{attribute addProperty BoxType "EL6201-0000-0017"}
{attribute addProperty Id "Slave_1_OutputsAT %Q*Slave_1_Outputs_44535924811Slave_2_OutputsAT %Q*Slave_2_Outputs_DA85B14E819Slave_3_OutputsAT %Q*Slave_3_Outputs_6031563F8117Slave_4_OutputsAT %Q*Slave_4_Outputs_A2C52F8B8125Slave_5_OutputsAT %Q*Slave_5_Outputs_502A55918133Slave_6_OutputsAT %Q*Slave_6_Outputs_564C8B0F8141Slave_7_OutputsAT %Q*Slave_7_Outputs_0A95F91A8149Slave_8_OutputsAT %Q*Slave_8_Outputs_C94C3BE28157Slave_9_OutputsAT %Q*Slave_9_Outputs_10CA7D998165Slave_10_OutputsAT %Q*Slave_10_Outputs_BCBE3A9D8173Slave_11_OutputsAT %Q*Slave_11_Outputs_22455BE68181Slave_12_OutputsAT %Q*Slave_12_Outputs_D1D6834F8189Slave_13_OutputsAT %Q*Slave_13_Outputs_D5DF10758197Slave_14_OutputsAT %Q*Slave_14_Outputs_41D7E34681105Slave_15_OutputsAT %Q*Slave_15_Outputs_5A42744581113Slave_16_OutputsAT %Q*Slave_16_Outputs_7177698381121Slave_17_OutputsAT %Q*Slave_17_Outputs_13B1B56F81129Slave_18_OutputsAT %Q*Slave_18_Outputs_11739BEB81137Slave_19_OutputsAT %Q*Slave_19_Outputs_5A6EF35981145Slave_20_OutputsAT %Q*Slave_20_Outputs_6270583781153Slave_21_OutputsAT %Q*Slave_21_Outputs_243B0FBE81161Slave_22_OutputsAT %Q*Slave_22_Outputs_2B83991D81169Slave_23_OutputsAT %Q*Slave_23_Outputs_88AC930781177Slave_24_OutputsAT %Q*Slave_24_Outputs_5EE1C1FB81185Slave_25_OutputsAT %Q*Slave_25_Outputs_6DA77E2C81193Slave_26_OutputsAT %Q*Slave_26_Outputs_8DCAE7C081201Slave_27_OutputsAT %Q*Slave_27_Outputs_EF0C3B2C81209Slave_28_OutputsAT %Q*Slave_28_Outputs_BE65F2CA81217Slave_29_OutputsAT %Q*Slave_29_Outputs_627166EC81225Slave_30_OutputsAT %Q*Slave_30_Outputs_FC69E36F81233Slave_31_OutputsAT %Q*Slave_31_Outputs_3BA48EB981241"}
{attribute addProperty CRC "1243080008"}
{attribute addProperty SizeInBites "248"}
{attribute addProperty SizeInBytes "31"}
TYPE ASI_Outputs_Device_4A17E548 :
STRUCT
	{attribute addProperty Name "Slave_1_Outputs"}
	Slave_1_Outputs AT %Q* : Slave_1_Outputs_44535924;
	{attribute addProperty Name "Slave_2_Outputs"}
	Slave_2_Outputs AT %Q* : Slave_2_Outputs_DA85B14E;
	{attribute addProperty Name "Slave_3_Outputs"}
	Slave_3_Outputs AT %Q* : Slave_3_Outputs_6031563F;
	{attribute addProperty Name "Slave_4_Outputs"}
	Slave_4_Outputs AT %Q* : Slave_4_Outputs_A2C52F8B;
	{attribute addProperty Name "Slave_5_Outputs"}
	Slave_5_Outputs AT %Q* : Slave_5_Outputs_502A5591;
	{attribute addProperty Name "Slave_6_Outputs"}
	Slave_6_Outputs AT %Q* : Slave_6_Outputs_564C8B0F;
	{attribute addProperty Name "Slave_7_Outputs"}
	Slave_7_Outputs AT %Q* : Slave_7_Outputs_0A95F91A;
	{attribute addProperty Name "Slave_8_Outputs"}
	Slave_8_Outputs AT %Q* : Slave_8_Outputs_C94C3BE2;
	{attribute addProperty Name "Slave_9_Outputs"}
	Slave_9_Outputs AT %Q* : Slave_9_Outputs_10CA7D99;
	{attribute addProperty Name "Slave_10_Outputs"}
	Slave_10_Outputs AT %Q* : Slave_10_Outputs_BCBE3A9D;
	{attribute addProperty Name "Slave_11_Outputs"}
	Slave_11_Outputs AT %Q* : Slave_11_Outputs_22455BE6;
	{attribute addProperty Name "Slave_12_Outputs"}
	Slave_12_Outputs AT %Q* : Slave_12_Outputs_D1D6834F;
	{attribute addProperty Name "Slave_13_Outputs"}
	Slave_13_Outputs AT %Q* : Slave_13_Outputs_D5DF1075;
	{attribute addProperty Name "Slave_14_Outputs"}
	Slave_14_Outputs AT %Q* : Slave_14_Outputs_41D7E346;
	{attribute addProperty Name "Slave_15_Outputs"}
	Slave_15_Outputs AT %Q* : Slave_15_Outputs_5A427445;
	{attribute addProperty Name "Slave_16_Outputs"}
	Slave_16_Outputs AT %Q* : Slave_16_Outputs_71776983;
	{attribute addProperty Name "Slave_17_Outputs"}
	Slave_17_Outputs AT %Q* : Slave_17_Outputs_13B1B56F;
	{attribute addProperty Name "Slave_18_Outputs"}
	Slave_18_Outputs AT %Q* : Slave_18_Outputs_11739BEB;
	{attribute addProperty Name "Slave_19_Outputs"}
	Slave_19_Outputs AT %Q* : Slave_19_Outputs_5A6EF359;
	{attribute addProperty Name "Slave_20_Outputs"}
	Slave_20_Outputs AT %Q* : Slave_20_Outputs_62705837;
	{attribute addProperty Name "Slave_21_Outputs"}
	Slave_21_Outputs AT %Q* : Slave_21_Outputs_243B0FBE;
	{attribute addProperty Name "Slave_22_Outputs"}
	Slave_22_Outputs AT %Q* : Slave_22_Outputs_2B83991D;
	{attribute addProperty Name "Slave_23_Outputs"}
	Slave_23_Outputs AT %Q* : Slave_23_Outputs_88AC9307;
	{attribute addProperty Name "Slave_24_Outputs"}
	Slave_24_Outputs AT %Q* : Slave_24_Outputs_5EE1C1FB;
	{attribute addProperty Name "Slave_25_Outputs"}
	Slave_25_Outputs AT %Q* : Slave_25_Outputs_6DA77E2C;
	{attribute addProperty Name "Slave_26_Outputs"}
	Slave_26_Outputs AT %Q* : Slave_26_Outputs_8DCAE7C0;
	{attribute addProperty Name "Slave_27_Outputs"}
	Slave_27_Outputs AT %Q* : Slave_27_Outputs_EF0C3B2C;
	{attribute addProperty Name "Slave_28_Outputs"}
	Slave_28_Outputs AT %Q* : Slave_28_Outputs_BE65F2CA;
	{attribute addProperty Name "Slave_29_Outputs"}
	Slave_29_Outputs AT %Q* : Slave_29_Outputs_627166EC;
	{attribute addProperty Name "Slave_30_Outputs"}
	Slave_30_Outputs AT %Q* : Slave_30_Outputs_FC69E36F;
	{attribute addProperty Name "Slave_31_Outputs"}
	Slave_31_Outputs AT %Q* : Slave_31_Outputs_3BA48EB9;
END_STRUCT
END_TYPE

(* stored: Version 1.2.0.0, ProductVersion 3.1.4024.9
   DUT ASI_Outputs_Device_4A17E548: Id {aebbd902-5a90-4e66-800a-e8b577f26c92} *)
